Fanuc KAREL source: ko00085.KL

-- PROVISIONAL review KL for V1013-1; original PC SHA256 2361328f41e7ab7de08c6d1272695ab34fcc016081f1b56479aafda2d26866c3
-- Incomplete behavior may be omitted. Consult companion uncertainty JSON. Do not deploy.
PROGRAM KO00085
%NOLOCKGROUP
BEGIN
  -- UNRESOLVED_PC offsets 5-12; opcodes 9D,23
  -- UNRESOLVED_PC offsets 17-69; opcodes 27,27,49,7E,AD,27,49,7E,AD,22,31,7E,4A
  -- UNRESOLVED_PC offsets 74-78; opcodes 7F
END KO00085
